PROGRAM prgComEffIO
VAR
	fbCom		: FB_MqttCommunicator_V2;
	
END_VAR


fbCom(
	bConnect:= TRUE, 
	strAuthKey:= 'EIO08031879806', 
	sUserName:= 'bc743937-b9db-4eca-8edf-ab66d553fcb7', 
	sUserPassword:= 'ae68774f-e424-481b-9a1e-cd1e957725b8', 
	eSavePositionCertificate:= eSavePositionOnPLC.ePostionHardDisk,  
	time_HeartBeat_sec:= T#15S, 
	bConnected=> , 
	bError=> , 
	hrErrorCode=> , 
	eConnectionState=> , 
	eErrorMessage_Out=> );

END_PROGRAM

(* stored: Version 1.1.0.1, ProductVersion 3.1.4024.12
   POU prgComEffIO: Id {cbcd318b-bf51-484c-bcaa-d6efcdf43fe3}, SpecialFunc None *)
